// TIA Portal V20 export
// export: Created 2025-12-01T14:57:26.7176803Z, ExportSetting None, DisplayName Totally Integrated Automation Portal, DisplayVersion V20 Update 3, DisplayName TIA Portal Openness, DisplayVersion V20 Update 3, DisplayName TIA Portal Version Control Interface, DisplayVersion V20 Update 3, DisplayName STEP 7 Professional, DisplayVersion V20 Update 3, DisplayName STEP 7 Safety, DisplayVersion V20 Update 2, DisplayName WinCC Basic/Comfort/Advanced, DisplayVersion V20 Update 3, DisplayName WinCC Professional, DisplayVersion V20 Update 3, DisplayName WinCC Unified, DisplayVersion V20 Update 3
FUNCTION "FC603_ResetQuimarox" : Void   // FC603, LAD
{ S7_Optimized_Access := 'TRUE' }
// stored: AutoNumber false, SetENOAutomatically false
   VAR_INPUT
      ID_Quimarox : UInt;
   END_VAR
   VAR_IN_OUT
      Maux_formateo : Bool;
   END_VAR
   VAR_TEMP
      contador : UInt;
      Mesa_quimarox : UInt;
   END_VAR
BEGIN

NETWORK
TITLE = Distribucion

      L     "DB600_ConfigQuimarox".Quimarox[#ID_Quimarox].datos_config.Numero_MesaAsociada;
      T     #Mesa_quimarox;

      SET;  // No hay que hacer nada
      AN    "DB902_Estado_ZonaMesa".EstadoMesas[#Mesa_quimarox].PerReset_CBx;
      AN    "DB902_Estado_ZonaMesa".EstadoMesas[#Mesa_quimarox].Resetear_CBx;
      JC    fin;

      SET;  // Reseteo --> Enviar eventos
      A     "DB902_Estado_ZonaMesa".EstadoMesas[#Mesa_quimarox].Resetear_CBx;
      AN    #Maux_formateo;
      JC    evento_QRES;

      SET;  // Activar Fin de Reset
      A     "DB902_Estado_ZonaMesa".EstadoMesas[#Mesa_quimarox].PerReset_CBx;
      JC    fin_reset;

      BE;


NETWORK
TITLE = En el proceso de reset, buscamos todos los peines que tengan datos y les escribimos el 503 para envio de mensajes
//==============================================================================================
evento_QRES:NOP   0;


      L     1;
      T     #contador;


bucle:NOP   0;

      SET;
      AN    "DB601_PeinesQuimarox".Quimarox[#ID_Quimarox].vagon[#contador].Carrier_Cargado;
      JC    siguiente;

// como tenemos carga, escribimos el evento que formatea el mensaje del reset

      L     "CTE_Evento_QRST";
      T     "DB601_PeinesQuimarox".Quimarox[#ID_Quimarox].vagon[#contador].EventoAGenerar;

// y pasamos a supervisar el siguiente vagon

//==============================================================================================
siguiente:NOP   0;  // comprobamos si hemos llegado al máximo de los vagones

      L     #contador;
      L     "DB600_ConfigQuimarox".Quimarox[#ID_Quimarox].datos_config.Numero_vagones;
      >=I;
      JC    fin_qres;

// si no hemos saltado es porque nos quedan vagones que revisar

      L     1;
      L     #contador;
      +I;
      T     #contador;

      JU    bucle;

fin_qres:SET;
      S     #Maux_formateo;
      BE;


//==============================================================================================

NETWORK
TITLE = generación del fin de reset
//==============================================================================================
fin_reset:NOP   0;

// para poder dar el fin de reset tenemos que asegurar que todos los mensajes QRES se han enviado

      L     1;
      T     #contador;

bucle2:NOP   0;

      L     "DB601_PeinesQuimarox".Quimarox[#ID_Quimarox].vagon[#contador].EventoAGenerar;
      L     0;
      <>I;
      JC    quedan_mensajes;

// si no hemos saltado es porque nos quedan vagones que revisar

      L     #contador;
      L     "DB600_ConfigQuimarox".Quimarox[#ID_Quimarox].datos_config.Numero_vagones;
      >=I;
      JC    da_fin_reset;


      L     1;
      L     #contador;
      +I;
      T     #contador;

      JU    bucle2;

quedan_mensajes:NOP   0;
      CLR;
      =     "DB900_Estado_Mesas".EstadoVI[#Mesa_quimarox].Fin_VI;
      BE;

da_fin_reset:SET;
      R     #Maux_formateo;
      =     "DB900_Estado_Mesas".EstadoVI[#Mesa_quimarox].Fin_VI;
      BE;


NETWORK
TITLE = 

fin:  SET;
      R     #Maux_formateo;
      =     "DB900_Estado_Mesas".EstadoVI[#Mesa_quimarox].Fin_VI;
      BE;



END_FUNCTION
